FUNCTION_BLOCK FB_Void
VAR_INPUT
END_VAR
VAR_OUTPUT
END_VAR
VAR
	pSequenceMaster : POINTER TO PVOID;
	fbConveyor : FB_Conveyor;
	fbVoidConveyor : FB_Conveyor;
	pConveyor : POINTER TO FB_Conveyor;
END_VAR

pSequenceMaster := ADR(fbConveyor);

pConveyor := pSequenceMaster;

END_FUNCTION_BLOCK

(* stored: Version 1.1.0.1, ProductVersion 3.1.4022.16
   POU FB_Void: Id {28d1cb9f-6a8b-4c41-a79a-d873346e878b}, SpecialFunc None *)
